TYPE ST_OEE :
STRUCT
	AmountOfSheets			 		: DINT;
	AmoundOfProductsSheets			: DINT;
	
END_STRUCT
END_TYPE

(* stored: Version 1.1.0.1, ProductVersion 3.1.4020.12
   DUT ST_OEE: Id {b4db3ab3-b08a-4c24-aa34-a235e14e3167} *)
